// TIA Portal V19 export
DATA_BLOCK "SyncNode"   // DB168
{ DB_Accessible_From_OPC_UA := 'FALSE' }
// stored: DBAccessibleFromOPCUA false, DBAccessibleFromWebserver false, InstanceOfName Unit.Em2.typeSyncNode, InstanceOfType UDT, Namespace Unit.Em2
"Unit.Em2.typeSyncNode"
   // VAR
   //    commands { ExternalWritable := 'False'} : Struct
   //       enableHpMotion : Bool;
   //    END_STRUCT;
   //    status { ExternalWritable := 'False'} : Struct
   //       busy : Bool;
   //       error : Bool;
   //    END_STRUCT;
   // END_VAR
BEGIN
END_DATA_BLOCK
